FUNCTION_BLOCK ListOfBytesTest EXTENDS TcUnit.FB_TestSuite
VAR
	staticArray : ARRAY [0..5] OF BYTE := [0, 1, 2, 3, 4, 5];
	listToTest : TwinCAT_OpenFramework_Collections.ListOfBytes;
END_VAR

LoadFromVariable();
GetAndSet();
Find();
Remove();
RemoveAt();
Resize();
Clear();

METHOD Clear
TEST(__POUNAME());

listToTest.Clear(TRUE);

AssertEquals_DINT(Expected := 0, Actual := listToTest._MemorySize, Message := 'Invalid memory size');
AssertEquals_DINT(Expected := 0, Actual := listToTest.Count, Message := 'Invalid byte count');

TEST_FINISHED();
END_METHOD

METHOD Find
VAR
	result : BOOL;
	index : DINT;
END_VAR
TEST(__POUNAME());

result := listToTest.Find(50, index => index);

AssertEquals_BOOL(Expected := TRUE, Actual := result, Message := 'Value not found');
AssertEquals_DINT(Expected := 5, Actual := index, Message := 'Wrong index of found element');
 
TEST_FINISHED();
END_METHOD

METHOD GetAndSet
VAR
	exceptionCode : __SYSTEM.ExceptionCode;
	errorMessage : TwinCAT_OpenFramework_Core.ERROR_MESSAGE;
END_VAR
TEST(__POUNAME());

listToTest.Clear();
listToTest.Append(staticArray[0]);
listToTest.Append(staticArray[1]);
listToTest.Append(staticArray[2]);
listToTest.Append(staticArray[3]);
listToTest.Append(staticArray[4]);
listToTest.Append(staticArray[5]); 

__TRY
	AssertEquals_BYTE(Expected := 5, Actual := listToTest.Get(5), Message := 'Invalid value received by Get');
	
	listToTest.Set(5, 50);

	AssertEquals_BYTE(Expected := 50, Actual := listToTest.Get(5), Message := 'Invalid value received by Get after Set');

	listToTest.Set(-1, 10);
__CATCH(exceptionCode)
	errorMessage := TwinCAT_OpenFramework_Core.ExceptionManager.GetLastException(exceptionCode).GetMessage();
	AssertEquals_STRING('Index is less then zero', WSTRING_TO_STRING(errorMessage), 'Wrong exception message');
__ENDTRY
 
TEST_FINISHED();
END_METHOD

METHOD LoadFromVariable
VAR
	exceptionCode : __SYSTEM.ExceptionCode;
	errorMessage : TwinCAT_OpenFramework_Core.ERROR_MESSAGE;
END_VAR
TEST(__POUNAME());

__TRY
	listToTest.LoadFromVariable(staticArray, 0);
	
	AssertEquals_DINT(Expected := TO_DINT(SIZEOF(staticArray)), Actual := listToTest.Count, Message := 'Data loading does not work properly');

	listToTest.LoadFromVariable(staticArray, -1);
__CATCH(exceptionCode)
	errorMessage := TwinCAT_OpenFramework_Core.ExceptionManager.GetLastException(exceptionCode).GetMessage();
	AssertEquals_STRING(Expected := 'Start index is less then zero', Actual := WSTRING_TO_STRING(errorMessage), Message := 'Wrong exception message');
__ENDTRY
 
TEST_FINISHED();
END_METHOD

METHOD Remove
TEST(__POUNAME());

listToTest.Clear();
listToTest.Append(staticArray[0]);
listToTest.Append(staticArray[1]);
listToTest.Append(staticArray[2]);
listToTest.Append(staticArray[3]);
listToTest.Append(staticArray[4]);
listToTest.Append(staticArray[5]); 

listToTest.Remove(2);

AssertEquals_DINT(Expected := 5, Actual := listToTest.Count, Message := 'Wrong array size');
AssertEquals_BYTE(Expected := 3, Actual := listToTest.Get(2), Message := 'Wrong element removing');
 
TEST_FINISHED();
END_METHOD

METHOD RemoveAt
TEST(__POUNAME());

listToTest.Clear();
listToTest.Append(staticArray[0]);
listToTest.Append(staticArray[1]);
listToTest.Append(staticArray[2]);
listToTest.Append(staticArray[3]);
listToTest.Append(staticArray[4]);
listToTest.Append(staticArray[5]); 

listToTest.RemoveAt(2, 2);

AssertEquals_DINT(Expected := 4, Actual := listToTest.Count, Message := 'Wrong array size');
AssertEquals_BYTE(Expected := 4, Actual := listToTest.Get(2), Message := 'Wrong element removing');
 
TEST_FINISHED();
END_METHOD

METHOD Resize
TEST(__POUNAME());

listToTest.Clear();
listToTest.Append(staticArray[0]);
listToTest.Append(staticArray[1]);
listToTest.Append(staticArray[2]);
listToTest.Append(staticArray[3]);
listToTest.Append(staticArray[4]);
listToTest.Append(staticArray[5]); 

listToTest.Resize(3);

AssertEquals_DINT(Expected := 3, Actual := listToTest.Count, Message := 'Wrong array size');
AssertEquals_BYTE(Expected := 2, Actual := listToTest.Get(2), Message := 'Wrong resizing');
 
TEST_FINISHED();
END_METHOD

END_FUNCTION_BLOCK

(* stored: Version 1.1.0.1, ProductVersion 3.1.4026.12
   POU ListOfBytesTest: Id {e0d457f1-7691-0ed2-12e6-5af4eb76f387}, SpecialFunc None
   Method Clear: Id {cc7b6cce-b32c-0e1b-3a5f-5cc4a98b3703}
   Method Find: Id {291851e1-364d-0b93-33e4-2a55e4f63de1}
   Method GetAndSet: Id {f3e83969-a851-0550-3369-b044cf3b7e76}
   Method LoadFromVariable: Id {257471d6-c1c9-0a5a-31cc-34a45c2c6e67}
   Method Remove: Id {43bf549b-b7ff-037c-02c7-57a820353e13}
   Method RemoveAt: Id {0da45385-69b4-029d-0187-17e53c4cff6e}
   Method Resize: Id {f041a7b6-9d21-0dc3-2bbd-11159243dede} *)
